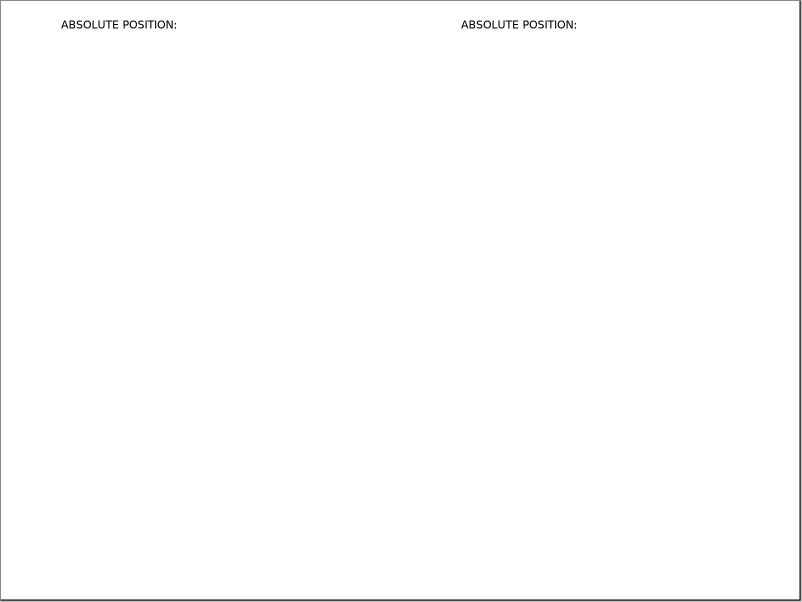
VISUALIZATION F30_Move_Additive  // 802x602
    Rectangle (0,0 800x600)
    Label (10,10 170x30), "ABSOLUTE POSITION:"
    Label (410,10 170x30), "ABSOLUTE POSITION:"
END_VISUALIZATION

(* stored: Version 1.1.0.1, ProductVersion 3.1.4022.7
   Visu F30_Move_Additive: Id {8681e353-6530-43cf-a5db-28408b088419} *)
